(* PLC project Water_Reserve_Control, Desconocido Sin nombre 1 *)
(* stored: creationDateTime 2024-11-13T10:20:43, modificationDateTime 2024-12-05T12:40:23 *)

PROGRAM Water_Control
  VAR
    Pool_Low_Level_Sensor AT %IX0.0 : BOOL;  (* Pools Level Sensor signal of min level. Zero indicates that level is under the minimun *)
    Tank_High_Level_Sensor AT %IX0.1 : BOOL;  (* Tank Level Sensor of miax level. State "1" indicates maximun level *)
    Water_Pump AT %QX0.0 : BOOL;  (* Pump state control output. High value turns on the motor *)
    Tank_Low_Level_Sensor AT %IX0.2 : BOOL;  (* Tank Level Sensor of min level. Zero indicates that level is under the minimun *)
    Automatic_Manual_Switch AT %IX0.3 : BOOL;  (* Automatic/Manual selector. State "0" is Manual mode and "1" Automatic mode *)
    Stop_Button AT %IX0.4 : BOOL;  (* Stop Push Button. If changes its value to "1" indicates stop de pump *)
    Start_Button AT %IX0.5 : BOOL;  (* Start Push Button. If changes its value to "1" indicates start de pump *)
  END_VAR

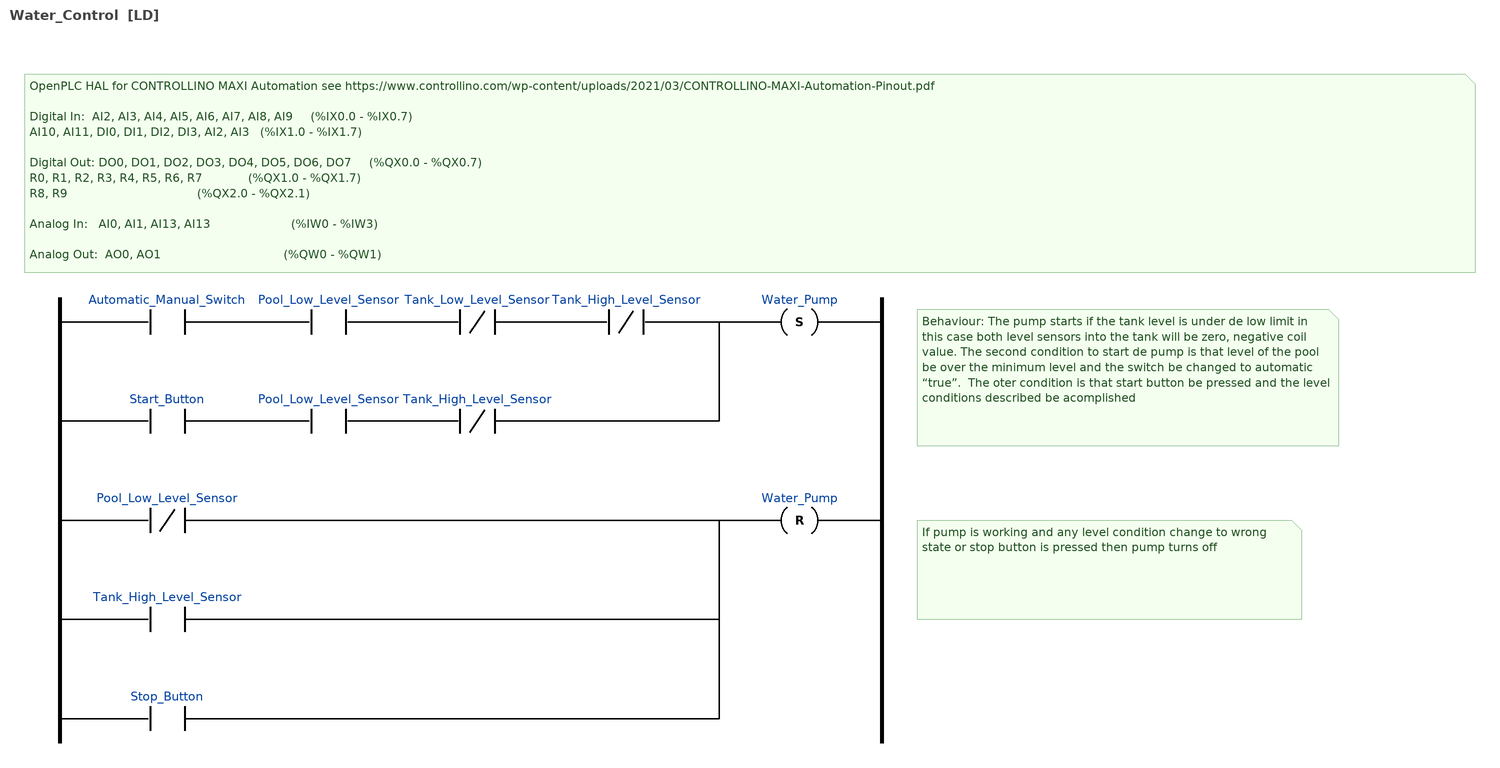
(* LD diagram, written out as Structured Text *)
(* OpenPLC HAL for CONTROLLINO MAXI Automation see https://www.controllino.com/wp-content/uploads/2021/03/CONTROLLINO-MAXI-Automation-Pinout.pdf

Digital In:  AI2, AI3, AI4, AI5, AI6, AI7, AI8, AI9     (%IX0.0 - %IX0.7)
             AI10, AI11, DI0, DI1, DI2, DI3, AI2, AI3   (%IX1.0 - %IX1.7)

Digital Out: DO0, DO1, DO2, DO3, DO4, DO5, DO6, DO7     (%QX0.0 - %QX0.7)
             R0, R1, R2, R3, R4, R5, R6, R7             (%QX1.0 - %QX1.7)
             R8, R9                                     (%QX2.0 - %QX2.1)

Analog In:   AI0, AI1, AI13, AI13                       (%IW0 - %IW3)

Analog Out:  AO0, AO1                                   (%QW0 - %QW1) *)
(* Behaviour: The pump starts if the tank level is under de low limit in this case both level sensors into the tank will be zero, negative coil value. The second condition to start de pump is that level of the pool be over the minimum level and the switch be changed to automatic “true”.  The oter condition is that start button be pressed and the level conditions described be acomplished *)
IF Automatic_Manual_Switch AND Pool_Low_Level_Sensor AND NOT Tank_Low_Level_Sensor AND NOT Tank_High_Level_Sensor OR Start_Button AND Pool_Low_Level_Sensor AND NOT Tank_High_Level_Sensor THEN Water_Pump := TRUE; END_IF;
IF NOT Pool_Low_Level_Sensor OR Stop_Button OR Tank_High_Level_Sensor THEN Water_Pump := FALSE; END_IF;
(* If pump is working and any level condition change to wrong state or stop button is pressed then pump turns off *)
END_PROGRAM

CONFIGURATION Config0
  RESOURCE Res0 ON PLC
    TASK task0(INTERVAL := T#20ms, PRIORITY := 0);
    PROGRAM instance0 WITH task0 : Water_Control;
  END_RESOURCE
END_CONFIGURATION
